TYPE ST_HMI_DataSourceConfig : 
STRUCT
	nID: DINT;
	sName: STRING(80);
	sDisplayName: STRING(80);
	nStreamCount: INT;
	aStreams: ARRAY [0..9] OF ST_HMI_DataSourceStream;
END_STRUCT
END_TYPE

(* stored: Version 1.1.0.1
   DUT ST_HMI_DataSourceConfig: Id 591b8b7c-35ab-429f-b607-fcd1511245d4 *)
